{attribute 'pack_mode' := '2'}
TYPE ST_R_Parameter :
STRUCT
  _nStart               : DINT := 901;
  _nCount               : DINT :=   4;
  _rValue               : ARRAY[0..MAX_R_PARA] OF LREAL;
END_STRUCT
END_TYPE

(* stored: Version 1.1.0.1, ProductVersion 3.1.4024.12
   DUT ST_R_Parameter: Id {aff9af41-9afb-094c-3fb2-8e7eab52ad07} *)
